DATA_BLOCK "ID_PE_Reject"
{ S7_Optimized_Access := 'TRUE' }
VERSION : 0.1
NON_RETAIN
"FB_PE_Reject"

BEGIN

END_DATA_BLOCK

